// TIA Portal project "Shift Registers" (V15.1)

(* hardware
DEVICE "S71500/ET200MP station_1"  S7-1500 station
   slot 0: "Rail_0"  Rack  6ES7 590-1***0-0AA0
   slot 0: "PM 190W 120/230VAC"  PM 190W 120/230VAC  6EP1333-4BA00
   slot 1: "PLC_1"  CPU 1516-3 PN/DP  6ES7 516-3AN01-0AB0  V2.6
      slot 3: "CPU display_1"  6ES7591-1BA00-0AA0
   slot 2: "DQ 32x24VDC/0.5A HF_1"  DQ 32x24VDC/0.5A HF  6ES7 522-1BL01-0AB0  V1.1
   slot 3: "DI 32x24VDC HF_1"  DI 32x24VDC HF  6ES7 521-1BL00-0AB0  V2.1
   slot 4: "AQ 4xU/I ST_1"  AQ 4xU/I ST  6ES7 532-5HD00-0AB0  V2.2
   slot 5: "AI 8xU/I/RTD/TC ST_1"  AI 8xU/I/RTD/TC ST  6ES7 531-7KF00-0AB0  V2.2
*)

// ===== PLC "PLC_1"  CPU 1516-3 PN/DP =====

VAR_GLOBAL   // PLC tag table "Full_Tag_Table"
   "Panel Emergency Stop" AT %I2.7 : Bool;
   "Start switch" AT %I0.2 : Bool;
   "Stop switch" AT %I0.3 : Bool;
   "Sort area IR" AT %I0.4 : Bool;
   "Sort Area Inductive" AT %I0.5 : Bool;
   "Sort Solenoid Sensor" AT %I0.6 : Bool;
   "Assembly Chute IR" AT %I0.7 : Bool;
   "Assembly Area Through Beam" AT %I1.1 : Bool;
   "Assembly Area Capacitor" AT %I1.2 : Bool;
   "Assembly Area Inductive" AT %I1.3 : Bool;
   "Reject Area IR" AT %I1.4 : Bool;
   "Reject Solenoid Sensor" AT %I1.5 : Bool;
   "Oven Through Beam" AT %I1.6 : Bool;
   "Loading Area Inductive" AT %I1.7 : Bool;
   "Chain Conveyor" AT %Q0.0 : Bool;
   "Sort Solenoid" AT %Q0.1 : Bool;
   "Reject Solenoid" AT %Q0.2 : Bool;
   "Rotary Solenoid" AT %Q0.3 : Bool;
   "Belt Conveyor Direction" AT %Q0.4 : Bool;
   "System Run_Green Lamp" AT %Q3.0 : Bool;
   "Sysyem Stop_Red Lamp" AT %Q3.2 : Bool;
   "Emergency stop" AT %I1.0 : Bool;
   "Ring Queue counter Full" AT %M4.0 : Bool;
   "Sort Solenoid error" AT %M4.3 : Bool;
   "Counter value" AT %MW0 : Int;
   "Reject Solenoid Error" AT %M4.7 : Bool;
   "HMI_Start" AT %M4.1 : Bool;
   "HMI_Stop" AT %M4.2 : Bool;
   "Counter Reset" AT %M4.4 : Bool;
   "Assembly Complete" AT %M4.5 : Bool;
   "Reset" AT %M4.6 : Bool;
END_VAR

DATA_BLOCK "Automatic_Conveyor_DB"   // DB1
{ S7_Optimized_Access := 'TRUE' }
VERSION : 0.1
// stored: InstanceOfName Automatic_Conveyor
"Automatic_Conveyor"
BEGIN
END_DATA_BLOCK

DATA_BLOCK "Sort Solenoid Active_DB"   // DB2
{ S7_Optimized_Access := 'TRUE' }
VERSION : 0.1
// stored: InstanceOfName Sort Solenoid Active
"Sort Solenoid Active"
BEGIN
END_DATA_BLOCK

DATA_BLOCK "Solenoids Error_DB"   // DB3
{ S7_Optimized_Access := 'TRUE' }
VERSION : 0.1
// stored: InstanceOfName Solenoids Error
"Solenoids Error"
BEGIN
END_DATA_BLOCK

DATA_BLOCK "Rotary Solenoid Active_DB"   // DB4
{ S7_Optimized_Access := 'TRUE' }
VERSION : 0.1
// stored: InstanceOfName Rotary Solenoid Active
"Rotary Solenoid Active"
BEGIN
END_DATA_BLOCK

DATA_BLOCK "Counting_DB"   // DB5
{ S7_Optimized_Access := 'TRUE' }
VERSION : 0.1
// stored: InstanceOfName Counting
"Counting"
BEGIN
END_DATA_BLOCK

DATA_BLOCK "Solenoids Error_DB_1"   // DB6
{ S7_Optimized_Access := 'TRUE' }
VERSION : 0.1
// stored: InstanceOfName Solenoids Error
"Solenoids Error"
BEGIN
END_DATA_BLOCK

DATA_BLOCK "Component Queue Handling_DB"   // DB7
{ S7_Optimized_Access := 'TRUE' }
VERSION : 0.1
// stored: InstanceOfName Component Queue Handling
"Component Queue Handling"
BEGIN
END_DATA_BLOCK

FUNCTION_BLOCK "Automatic_Conveyor"   // FB1, LAD
TITLE = Conveyors Automatic
{ S7_Optimized_Access := 'TRUE' }
VERSION : 0.1
   VAR_INPUT
      "Start Switch" : Bool;
      "Stop Switch" : Bool;
      "Emergency Stop" : Bool;
      "Panel Emergency Stop" : Bool;
      "Sort Solenoid Error" : Bool;
      "Reject Solenoid Error" : Bool;
      "Assembly Done" : Bool;
      Reset : Bool;
   END_VAR
   VAR_OUTPUT
      "System Enable_OK" : Bool;
      "System Enable_not_OK" : Bool;
      "Chain Conveyor" : Bool;
      "Belt Conveyor" : Bool;
   END_VAR
   VAR
      Memory_Automatic_Start_Stop : Bool;
   END_VAR
BEGIN

REGION Network 1: System Enable_OK and Conveyors run
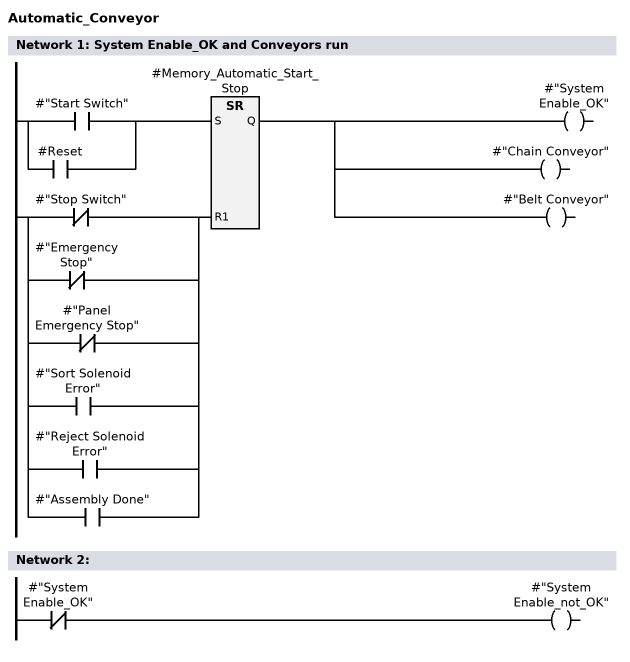
   RUNG wire#powerrail
      Contact( #"Start Switch" )
      wire#w1
      S_SR(operand := #Memory_Automatic_Start_Stop, r1 := wire#w2)
      wire#w3
      Coil( #"System Enable_OK" )
   END_RUNG
   RUNG wire#powerrail
      Contact( #Reset )
   END_RUNG wire#w1
   RUNG wire#powerrail
      I_Contact( #"Stop Switch" )
   END_RUNG wire#w2
   RUNG wire#powerrail
      I_Contact( #"Emergency Stop" )
   END_RUNG wire#w2
   RUNG wire#powerrail
      I_Contact( #"Panel Emergency Stop" )
   END_RUNG wire#w2
   RUNG wire#powerrail
      Contact( #"Sort Solenoid Error" )
   END_RUNG wire#w2
   RUNG wire#powerrail
      Contact( #"Reject Solenoid Error" )
   END_RUNG wire#w2
   RUNG wire#powerrail
      Contact( #"Assembly Done" )
   END_RUNG wire#w2
   RUNG wire#w3
      Coil( #"Chain Conveyor" )
   END_RUNG
   RUNG wire#w3
      Coil( #"Belt Conveyor" )
   END_RUNG
   // the same network as SCL:
   IF #"Start Switch" OR #Reset THEN
       #Memory_Automatic_Start_Stop := TRUE;   // SR flip-flop
   END_IF;
   IF NOT #"Stop Switch" OR NOT #"Emergency Stop" OR NOT #"Panel Emergency Stop" OR #"Sort Solenoid Error" OR #"Reject Solenoid Error" OR #"Assembly Done" THEN
       #Memory_Automatic_Start_Stop := FALSE;
   END_IF;
   #"System Enable_OK" := #Memory_Automatic_Start_Stop;
   #"Chain Conveyor" := #Memory_Automatic_Start_Stop;
   #"Belt Conveyor" := #Memory_Automatic_Start_Stop;
END_REGION

REGION Network 2
   RUNG wire#powerrail
      I_Contact( #"System Enable_OK" )
      Coil( #"System Enable_not_OK" )
   END_RUNG
   // the same network as SCL:
   #"System Enable_not_OK" := NOT #"System Enable_OK";
END_REGION
END_FUNCTION_BLOCK

FUNCTION_BLOCK "Sort Solenoid Active"   // FB2, LAD
TITLE = Sort Solenoid Active
{ S7_Optimized_Access := 'TRUE' }
VERSION : 0.1
   VAR_INPUT
      "Sort Area IR" : Bool;
      "Sort Area Inductive" : Bool;
      "Ring Counter Full" : Bool;
   END_VAR
   VAR_OUTPUT
      "Sort Solenoid" : Bool;
   END_VAR
   VAR
      "Component Pass Delay" : Bool;
      "SR_Sort Solenoid on Timer" : Bool;
      "SR_Component Pass Delay" : Bool;
      IEC_Timer_0_Instance : TON_TIME;
      IEC_Timer_0_Instance_2 : TON_TIME;
   END_VAR
BEGIN

REGION Network 1: Sort Solenoid Active if Plastic Ring Present
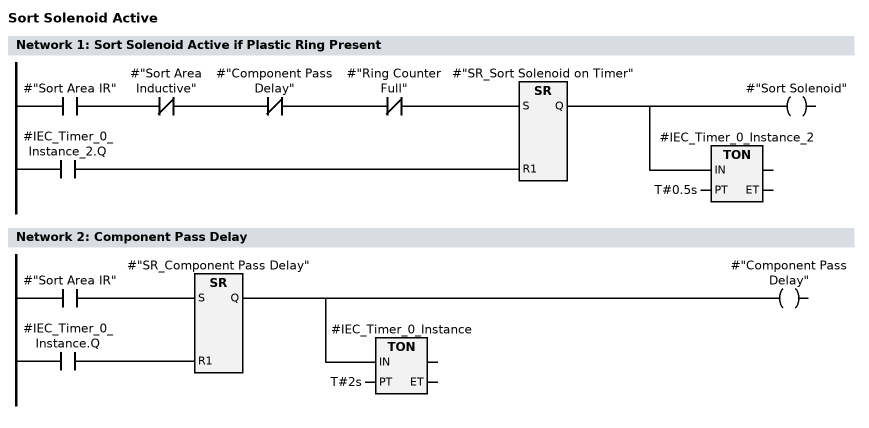
   IF #"Sort Area IR" AND NOT #"Sort Area Inductive" AND NOT #"Component Pass Delay" AND NOT #"Ring Counter Full" THEN
       #"SR_Sort Solenoid on Timer" := TRUE;   // SR flip-flop
   END_IF;
   IF #IEC_Timer_0_Instance_2.Q THEN #"SR_Sort Solenoid on Timer" := FALSE; END_IF;
   #"Sort Solenoid" := #"SR_Sort Solenoid on Timer";
   #IEC_Timer_0_Instance_2(IN := #"SR_Sort Solenoid on Timer", PT := T#0.5s);   // TON
END_REGION

REGION Network 2: Component Pass Delay
   IF #"Sort Area IR" THEN
       #"SR_Component Pass Delay" := TRUE;   // SR flip-flop
   END_IF;
   IF #IEC_Timer_0_Instance.Q THEN #"SR_Component Pass Delay" := FALSE; END_IF;
   #"Component Pass Delay" := #"SR_Component Pass Delay";
   #IEC_Timer_0_Instance(IN := #"SR_Component Pass Delay", PT := T#2s);   // TON
END_REGION
END_FUNCTION_BLOCK

FUNCTION_BLOCK "Solenoids Error"   // FB3, LAD
TITLE = Solenoid Error - Closed Loop Control
{ S7_Optimized_Access := 'TRUE' }
VERSION : 0.1
   VAR_INPUT
      "Solenoid on" : Bool;
      "Solenoid sensor" : Bool;
   END_VAR
   VAR_OUTPUT
      "Solenoid Error" : Bool;
   END_VAR
   VAR
      "Hold off delay" : Bool;
      IEC_Timer_0_Instance : TON_TIME;
   END_VAR
BEGIN

REGION Network 1: Solenoid Error
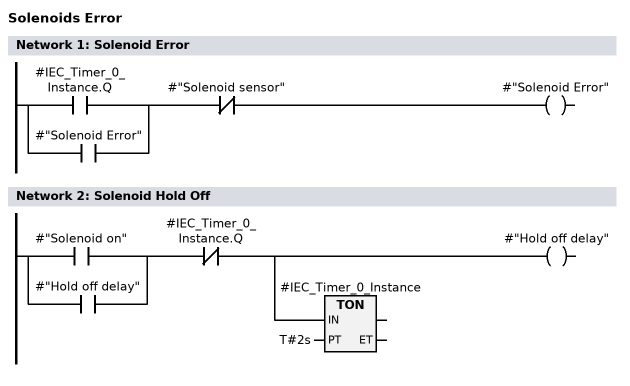
   RUNG wire#powerrail
      Contact( #IEC_Timer_0_Instance.Q )
      wire#w1
      I_Contact( #"Solenoid sensor" )
      Coil( #"Solenoid Error" )
   END_RUNG
   RUNG wire#powerrail
      Contact( #"Solenoid Error" )
   END_RUNG wire#w1
   // the same network as SCL:
   #"Solenoid Error" := (#IEC_Timer_0_Instance.Q OR #"Solenoid Error") AND NOT #"Solenoid sensor";
END_REGION

REGION Network 2: Solenoid Hold Off
   #"Hold off delay" := (#"Solenoid on" OR #"Hold off delay") AND NOT #IEC_Timer_0_Instance.Q;
   #IEC_Timer_0_Instance(IN := #"Hold off delay", PT := T#2s);   // TON
END_REGION
END_FUNCTION_BLOCK

FUNCTION_BLOCK "Counting"   // FB4, LAD
TITLE = Counting
{ S7_Optimized_Access := 'TRUE' }
VERSION : 0.1
// Incremental and Decremental counting
   VAR_INPUT
      "Sort Solenoid" : Bool;
      "Rotary Solenoid" : Bool;
   END_VAR
   VAR_OUTPUT
      "Ring Queue counter full" : Bool;
      "Counter Value" : Int;
   END_VAR
   VAR RETAIN
      IEC_Counter_0_Instance : CTUD_INT;
   END_VAR
BEGIN

REGION Network 1: Counting
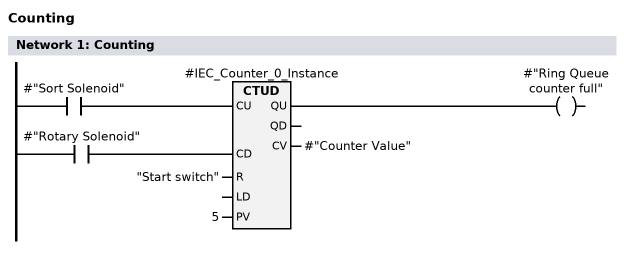
   #IEC_Counter_0_Instance(CU := #"Sort Solenoid",   // CTUD
                           CD := #"Rotary Solenoid",
                           R := "Start switch",
                           PV := 5,
                           CV => #"Counter Value");
   #"Ring Queue counter full" := #IEC_Counter_0_Instance.QU;
END_REGION
END_FUNCTION_BLOCK

FUNCTION_BLOCK "Rotary Solenoid Active"   // FB5, LAD
TITLE = Rotary Solenoid Active
{ S7_Optimized_Access := 'TRUE' }
VERSION : 0.1
   VAR_INPUT
      "Rotary Area IR" : Bool;
   END_VAR
   VAR_OUTPUT
      "Rotary Solenoid" : Bool;
   END_VAR
   VAR
      "SR_Component Pass Delay" : Bool;
      "Component Pass Delay" : Bool;
      IEC_Timer_0_Instance : TON_TIME;
      IEC_Timer_0_Instance_2 : TON_TIME;
      "SR Rotary Solenoid on Timer" : Bool;
      IEC_Timer_0_Instance_1 : TON_TIME;
   END_VAR
BEGIN

REGION Network 1: Rotary Solenoid Activation
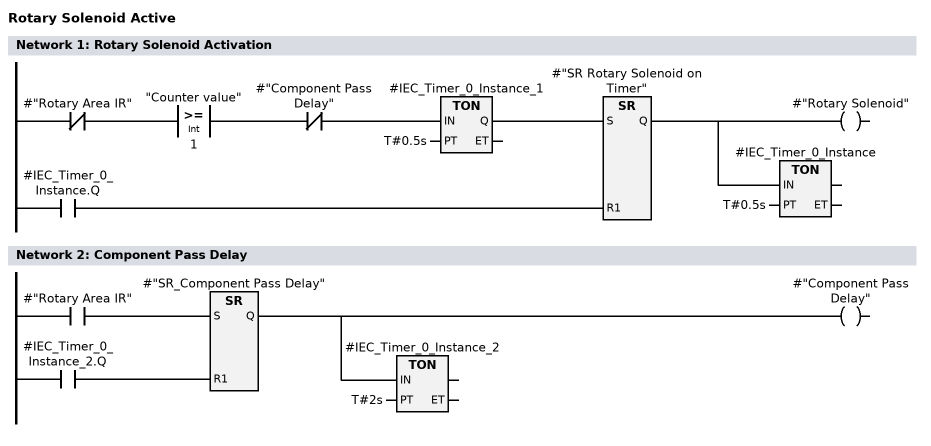
   #IEC_Timer_0_Instance_1(IN := NOT #"Rotary Area IR" AND ("Counter value" >= 1) AND NOT #"Component Pass Delay",   // TON
                           PT := T#0.5s);
   IF #IEC_Timer_0_Instance_1.Q THEN
       #"SR Rotary Solenoid on Timer" := TRUE;   // SR flip-flop
   END_IF;
   IF #IEC_Timer_0_Instance.Q THEN #"SR Rotary Solenoid on Timer" := FALSE; END_IF;
   #"Rotary Solenoid" := #"SR Rotary Solenoid on Timer";
   #IEC_Timer_0_Instance(IN := #"SR Rotary Solenoid on Timer", PT := T#0.5s);   // TON
END_REGION

REGION Network 2: Component Pass Delay
   IF #"Rotary Area IR" THEN
       #"SR_Component Pass Delay" := TRUE;   // SR flip-flop
   END_IF;
   IF #IEC_Timer_0_Instance_2.Q THEN #"SR_Component Pass Delay" := FALSE; END_IF;
   #"Component Pass Delay" := #"SR_Component Pass Delay";
   #IEC_Timer_0_Instance_2(IN := #"SR_Component Pass Delay", PT := T#2s);   // TON
END_REGION
END_FUNCTION_BLOCK

FUNCTION_BLOCK "Component Queue Handling"   // FB6, LAD
TITLE = Component Queue Handling
{ S7_Optimized_Access := 'TRUE' }
VERSION : 0.1
   VAR_INPUT
      "Start Switch" : Bool;
      "Assembly Area Capacitive" : Bool;
      "Assembly Area Inductive" : Bool;
      "Reject Area IR" : Bool;
      "Assembly Area Through Beam" : Bool;
   END_VAR
   VAR_OUTPUT
      "Reject Solenoid" : Bool;
      "Assembly Done" : Bool;
      Reset : Bool;
   END_VAR
   VAR
      "Pointer Register" : Word;
      "Data Register" : Word;
      "SHL Memory" : Bool;
      "SHR Memory" : Bool;
      "And Result" : Word;
      SR_Reject : Bool;
      IEC_Timer_0_Instance : TON_TIME;
      "Assembly Complete" : Bool;
      IEC_Timer_0_Instance_1 : TON_TIME;
      "SR_Assembly Done" : Bool;
      IEC_Timer_0_Instance_2 : TON_TIME;
      SR_Stop : Bool;
      SR_Reset : Bool;
      IEC_Timer_0_Instance_3 : TON_TIME;
      IEC_Timer_0_Instance_4 : TON_TIME;
      IEC_Timer_0_Instance_5 : TON_TIME;
      SR_Inductive : Bool;
      IEC_Timer_0_Instance_6 : TON_TIME;
      IEC_Timer_0_Instance_7 : TON_TIME;
      IEC_Timer_0_Instance_8 : TON_TIME;
   END_VAR
   VAR_TEMP   // added for the SCL form of the ladder/FBD networks
      _w1 : Bool;
   END_VAR
BEGIN

REGION Network 1: Data and pointer register
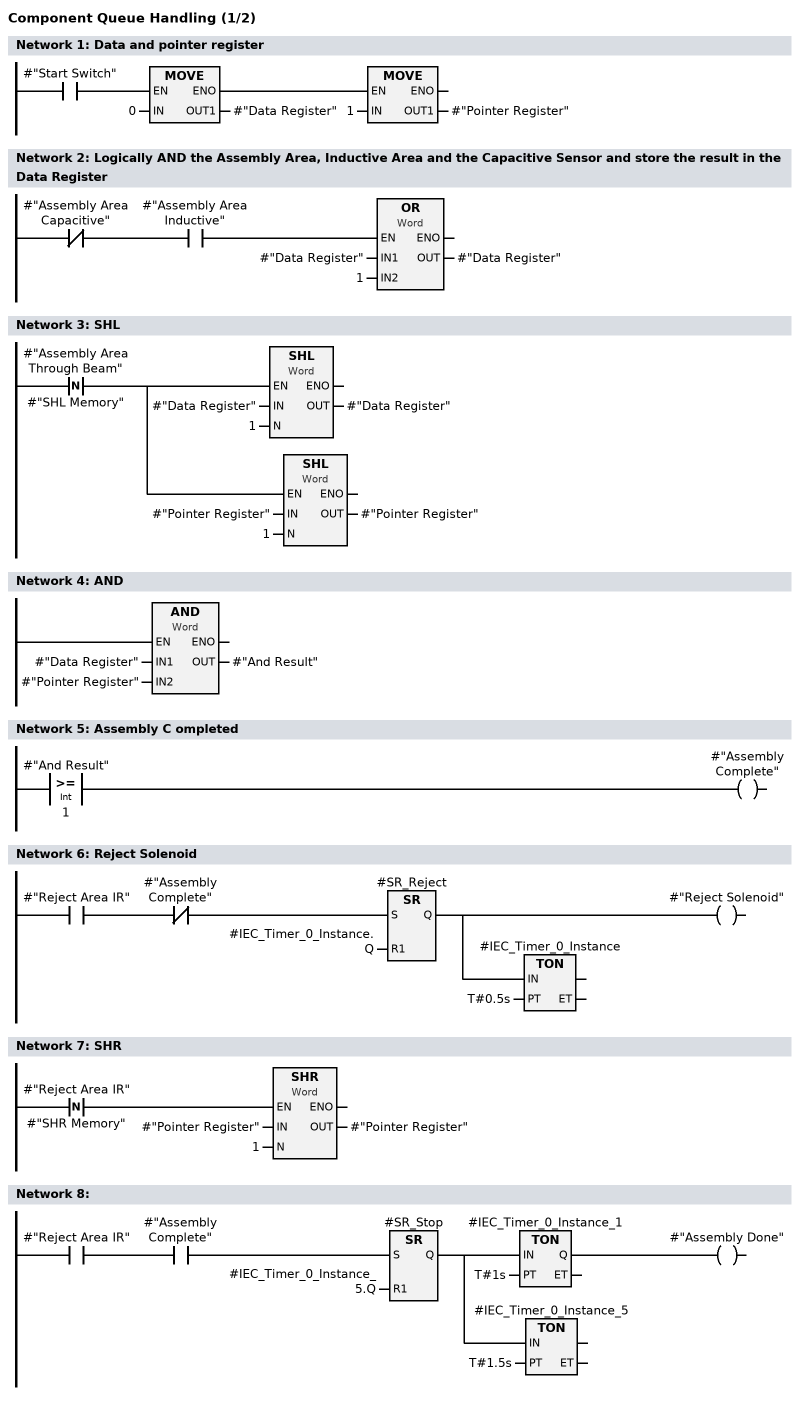
   RUNG wire#powerrail
      Contact( #"Start Switch" )
      Move(in := 0, out1 => #"Data Register")
      Move(in := 1, out1 => #"Pointer Register")
   END_RUNG
   // the same network as SCL:
   IF #"Start Switch" THEN
       #"Data Register" := 0;
       #"Pointer Register" := 1;
   END_IF;
END_REGION

REGION Network 2: Logically AND the Assembly Area, Inductive Area and the Capacitive Sensor and store the result in the Data Register
   IF NOT #"Assembly Area Capacitive" AND #"Assembly Area Inductive" THEN
       #"Data Register" := #"Data Register" OR 1;
   END_IF;
END_REGION

REGION Network 3: SHL
   RUNG wire#powerrail
      N_Contact(operand := #"Assembly Area Through Beam", bit := #"SHL Memory")
      wire#w1
      { S7_Templates := "SrcType := Word" } Shl(in := #"Data Register", n := 1, out => #"Data Register")
   END_RUNG
   RUNG wire#w1
      { S7_Templates := "SrcType := Word" } Shl(in := #"Pointer Register", n := 1, out => #"Pointer Register")
   END_RUNG
   // the same network as SCL:
   #_w1 := NOT #"Assembly Area Through Beam" AND #"SHL Memory";   // falling edge of #"Assembly Area Through Beam"
   #"SHL Memory" := #"Assembly Area Through Beam";
   IF #_w1 THEN
       #"Data Register" := SHL(IN := #"Data Register", N := 1);
       #"Pointer Register" := SHL(IN := #"Pointer Register", N := 1);
   END_IF;
END_REGION

REGION Network 4: AND
   RUNG wire#powerrail
      { S7_Templates := "SrcType := Word" } And(in1 := #"Data Register", in2 := #"Pointer Register", out => #"And Result")
   END_RUNG
   // the same network as SCL:
   #"And Result" := #"Data Register" AND #"Pointer Register";
END_REGION

REGION Network 5: Assembly C ompleted
   RUNG wire#powerrail
      { S7_Templates := "SrcType := Int" } GE_Contact(in1 := #"And Result", in2 := 1)
      Coil( #"Assembly Complete" )
   END_RUNG
   // the same network as SCL:
   #"Assembly Complete" := #"And Result" >= 1;
END_REGION

REGION Network 6: Reject Solenoid
   IF #"Reject Area IR" AND NOT #"Assembly Complete" THEN
       #SR_Reject := TRUE;   // SR flip-flop
   END_IF;
   IF #IEC_Timer_0_Instance.Q THEN #SR_Reject := FALSE; END_IF;
   #"Reject Solenoid" := #SR_Reject;
   #IEC_Timer_0_Instance(IN := #SR_Reject, PT := T#0.5s);   // TON
END_REGION

REGION Network 7: SHR
   RUNG wire#powerrail
      N_Contact(operand := #"Reject Area IR", bit := #"SHR Memory")
      { S7_Templates := "SrcType := Word" } Shr(in := #"Pointer Register", n := 1, out => #"Pointer Register")
   END_RUNG
   // the same network as SCL:
   #_w1 := NOT #"Reject Area IR" AND #"SHR Memory";   // falling edge of #"Reject Area IR"
   #"SHR Memory" := #"Reject Area IR";
   IF #_w1 THEN #"Pointer Register" := SHR(IN := #"Pointer Register", N := 1); END_IF;
END_REGION

REGION Network 8
   IF #"Reject Area IR" AND #"Assembly Complete" THEN
       #SR_Stop := TRUE;   // SR flip-flop
   END_IF;
   IF #IEC_Timer_0_Instance_5.Q THEN #SR_Stop := FALSE; END_IF;
   #IEC_Timer_0_Instance_1(IN := #SR_Stop, PT := T#1s);   // TON
   #"Assembly Done" := #IEC_Timer_0_Instance_1.Q;
   #IEC_Timer_0_Instance_5(IN := #SR_Stop, PT := T#1.5s);   // TON
END_REGION

REGION Network 9
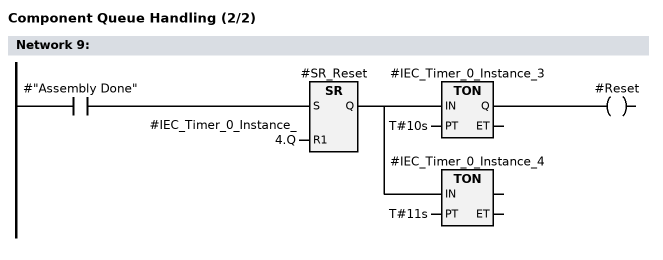
   IF #"Assembly Done" THEN
       #SR_Reset := TRUE;   // SR flip-flop
   END_IF;
   IF #IEC_Timer_0_Instance_4.Q THEN #SR_Reset := FALSE; END_IF;
   #IEC_Timer_0_Instance_3(IN := #SR_Reset, PT := T#10s);   // TON
   #Reset := #IEC_Timer_0_Instance_3.Q;
   #IEC_Timer_0_Instance_4(IN := #SR_Reset, PT := T#11s);   // TON
END_REGION
END_FUNCTION_BLOCK

ORGANIZATION_BLOCK "Main"   // OB1, LAD, ProgramCycle
TITLE = "Main Program Sweep (Cycle)"
{ S7_Optimized_Access := 'TRUE' }
VERSION : 0.1
   VAR_INPUT
      Initial_Call : Bool;   // Initial call of this OB
      Remanence : Bool;   // =True, if remanent data are available
   END_VAR
BEGIN

REGION Network 1: System run ok and conveyors start
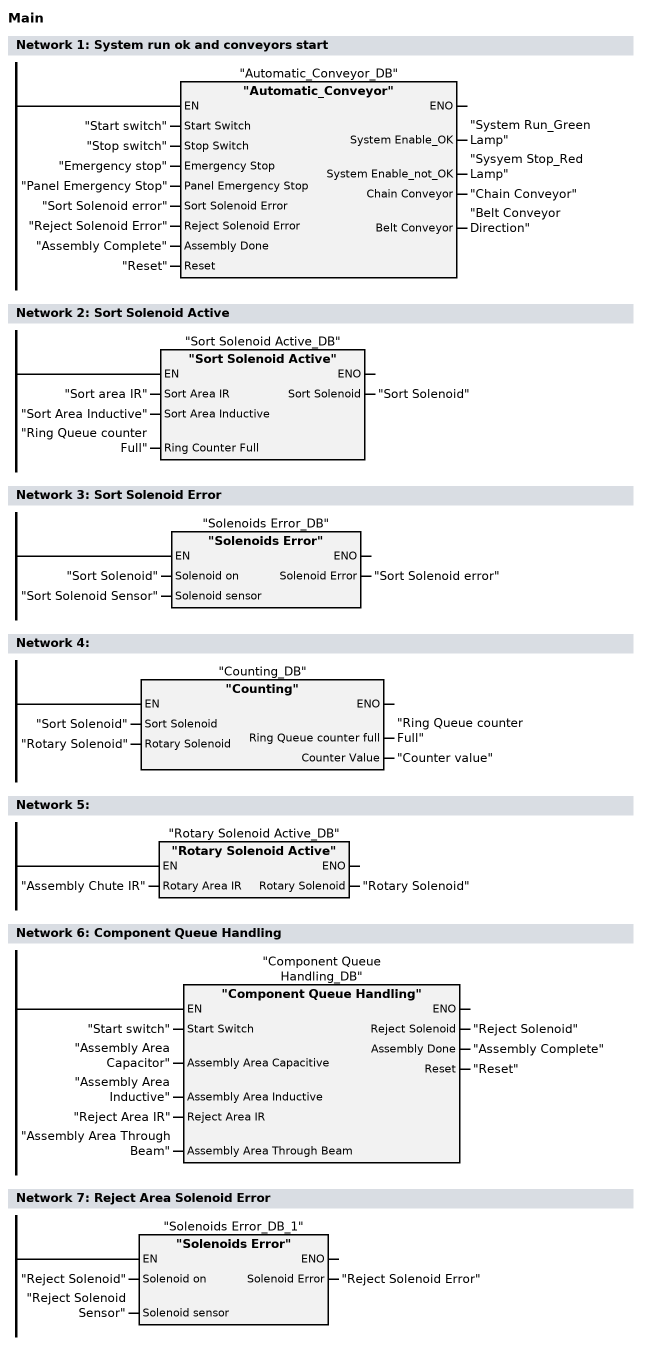
   RUNG wire#powerrail
      "Automatic_Conveyor_DB"("Start Switch" := "Start switch", "Stop Switch" := "Stop switch", "Emergency Stop" := "Emergency stop", "Panel Emergency Stop" := "Panel Emergency Stop", "Sort Solenoid Error" := "Sort Solenoid error", "Reject Solenoid Error" := "Reject Solenoid Error", "Assembly Done" := "Assembly Complete", Reset := "Reset", "System Enable_OK" => "System Run_Green Lamp", "System Enable_not_OK" => "Sysyem Stop_Red Lamp", "Chain Conveyor" => "Chain Conveyor", "Belt Conveyor" => "Belt Conveyor Direction")
   END_RUNG
   // the same network as SCL:
   "Automatic_Conveyor_DB"("Start Switch" := "Start switch",   // "Automatic_Conveyor"
                           "Stop Switch" := "Stop switch",
                           "Emergency Stop" := "Emergency stop",
                           "Panel Emergency Stop" := "Panel Emergency Stop",
                           "Sort Solenoid Error" := "Sort Solenoid error",
                           "Reject Solenoid Error" := "Reject Solenoid Error",
                           "Assembly Done" := "Assembly Complete",
                           Reset := "Reset",
                           "System Enable_OK" => "System Run_Green Lamp",
                           "System Enable_not_OK" => "Sysyem Stop_Red Lamp",
                           "Chain Conveyor" => "Chain Conveyor",
                           "Belt Conveyor" => "Belt Conveyor Direction");
END_REGION

REGION Network 2: Sort Solenoid Active
   RUNG wire#powerrail
      "Sort Solenoid Active_DB"("Sort Area IR" := "Sort area IR", "Sort Area Inductive" := "Sort Area Inductive", "Ring Counter Full" := "Ring Queue counter Full", "Sort Solenoid" => "Sort Solenoid")
   END_RUNG
   // the same network as SCL:
   "Sort Solenoid Active_DB"("Sort Area IR" := "Sort area IR",   // "Sort Solenoid Active"
                           "Sort Area Inductive" := "Sort Area Inductive",
                           "Ring Counter Full" := "Ring Queue counter Full",
                           "Sort Solenoid" => "Sort Solenoid");
END_REGION

REGION Network 3: Sort Solenoid Error
   RUNG wire#powerrail
      "Solenoids Error_DB"("Solenoid on" := "Sort Solenoid", "Solenoid sensor" := "Sort Solenoid Sensor", "Solenoid Error" => "Sort Solenoid error")
   END_RUNG
   // the same network as SCL:
   "Solenoids Error_DB"("Solenoid on" := "Sort Solenoid",   // "Solenoids Error"
                        "Solenoid sensor" := "Sort Solenoid Sensor",
                        "Solenoid Error" => "Sort Solenoid error");
END_REGION

REGION Network 4
   RUNG wire#powerrail
      "Counting_DB"("Sort Solenoid" := "Sort Solenoid", "Rotary Solenoid" := "Rotary Solenoid", "Ring Queue counter full" => "Ring Queue counter Full", "Counter Value" => "Counter value")
   END_RUNG
   // the same network as SCL:
   "Counting_DB"("Sort Solenoid" := "Sort Solenoid",   // "Counting"
                 "Rotary Solenoid" := "Rotary Solenoid",
                 "Ring Queue counter full" => "Ring Queue counter Full",
                 "Counter Value" => "Counter value");
END_REGION

REGION Network 5
   RUNG wire#powerrail
      "Rotary Solenoid Active_DB"("Rotary Area IR" := "Assembly Chute IR", "Rotary Solenoid" => "Rotary Solenoid")
   END_RUNG
   // the same network as SCL:
   "Rotary Solenoid Active_DB"("Rotary Area IR" := "Assembly Chute IR", "Rotary Solenoid" => "Rotary Solenoid");   // "Rotary Solenoid Active"
END_REGION

REGION Network 6: Component Queue Handling
   RUNG wire#powerrail
      "Component Queue Handling_DB"("Start Switch" := "Start switch", "Assembly Area Capacitive" := "Assembly Area Capacitor", "Assembly Area Inductive" := "Assembly Area Inductive", "Reject Area IR" := "Reject Area IR", "Assembly Area Through Beam" := "Assembly Area Through Beam", "Reject Solenoid" => "Reject Solenoid", "Assembly Done" => "Assembly Complete", Reset => "Reset")
   END_RUNG
   // the same network as SCL:
   "Component Queue Handling_DB"("Start Switch" := "Start switch",   // "Component Queue Handling"
                           "Assembly Area Capacitive" := "Assembly Area Capacitor",
                           "Assembly Area Inductive" := "Assembly Area Inductive",
                           "Reject Area IR" := "Reject Area IR",
                           "Assembly Area Through Beam" := "Assembly Area Through Beam",
                           "Reject Solenoid" => "Reject Solenoid",
                           "Assembly Done" => "Assembly Complete",
                           Reset => "Reset");
END_REGION

REGION Network 7: Reject Area Solenoid Error
   RUNG wire#powerrail
      "Solenoids Error_DB_1"("Solenoid on" := "Reject Solenoid", "Solenoid sensor" := "Reject Solenoid Sensor", "Solenoid Error" => "Reject Solenoid Error")
   END_RUNG
   // the same network as SCL:
   "Solenoids Error_DB_1"("Solenoid on" := "Reject Solenoid",   // "Solenoids Error"
                          "Solenoid sensor" := "Reject Solenoid Sensor",
                          "Solenoid Error" => "Reject Solenoid Error");
END_REGION
END_ORGANIZATION_BLOCK